Fanuc KAREL source: compact_preamble.KL

PROGRAM KB00199
%NOLOCKGROUP
VAR
P1 : FILE
P2 : STRING[80]
P3:INTEGER
P4:BOOLEAN
P5:INTEGER
P6:INTEGER
BEGIN
P2='A'
P3=1
P4=TRUE
P5=1
P6=1
XML_ADDTAG(P1,P2,P3,P4,P5,P6)
END KB00199
